Staubli VAL3: getDBsize.pgx

public program getDBsize(num x_nDBnumber, num& x_nSize)
  local num l_nLength
  local num l_nS7_BI[37]
begin

  call setLastError(nNoErrors)
  x_nSize=0

  //setup the telegram
  getData("nS7_BI", l_nS7_BI)

  l_nS7_BI[31]=round((x_nDBnumber/10000)+48)
  x_nDBnumber=round(x_nDBnumber%10000)

  l_nS7_BI[32]=round((x_nDBnumber/1000)+48)
  x_nDBnumber=round(x_nDBnumber%1000)

  l_nS7_BI[33]=round((x_nDBnumber/100)+48)
  x_nDBnumber=round(x_nDBnumber%100)

  l_nS7_BI[34]=round((x_nDBnumber/10)+48)
  x_nDBnumber=round(x_nDBnumber%10)

  l_nS7_BI[35]=round((x_nDBnumber)+48)

  call sendPacket(l_nS7_BI, size(l_nS7_BI))
  if nLastError==nNoErrors
    call recvISOpacket(l_nLength)
    //26 is the minimum expected
    if l_nLength>=26
      //if ((PDU.H[37]==0x00) && (PDU.H[38]==0x00) && (PDU.H[39]==0xFF))
      if PDU.S7telegram.DATA[2]==0 or PDU.S7telegram.DATA[3]==0 or PDU.S7telegram.DATA[4]==255
        x_nSize=PDU.S7telegram.DATA[48]
        x_nSize=x_nSize*power(2,8)+PDU.S7telegram.DATA[49]
      else
        call setLastError(nErrS7Func)
      endIf
    else
      call setLastError(nErrISOInvPDU)
    endIf
  else
    call setLastError(nErrTCPSend)
  endIf

end
